Universal Robots PolyScope program: rtde_control_loop.urp

Program rtde_control_loop (installation=default directory=/programs/usbdisk createdIn=3.2.19275 lastSavedIn=0.0.0 robotSerialNumber=20195001564)
Calibrated DH parameters: a=[0.000053, -0.575316, -0.491508, -0.00015, 0.000016, 0]; d=[0.181047, 73.792979, -575.127925, 501.508986, 0.1198, 0.115548]; alpha=[1.570273, 0.002844, 0.000581, 1.569979, -1.569422, 0]; deltaTheta=[-0.000001, 0.349752, 5.398781, 0.534651, 0.000006, 0]
InitVariablesNode
BeforeStart
  setp := Joint_6_name
  SuppressedNode
    Script: rtde_set_watchdog("input_int_register_0", 1, "PAUSE")
Robot Program (runOnlyOnce=false)
  Script: write_output_integer_register(0, 0)
  Wait Sleep waitTime=0.01
  MoveL speed 250 mm/s, acceleration 1200 mm/s^2 (useActiveTCP=true) feature=Base
    Waypoint Variable (Variable): variable=setp
  Script: write_output_integer_register(0, 1)
  Wait Sleep waitTime=0.01
Thread Thread_1 (runOnlyOnce=false)
  setp := Joint_6_name
  Loop Forever
    tmp := p[0,0,0,0,0,0]
    Script: tmp[0] = read_input_float_register(0)
    Script: tmp[1] = read_input_float_register(1)
    Script: tmp[2] = read_input_float_register(2)
    Script: tmp[3] = read_input_float_register(3)
    Script: tmp[4] = read_input_float_register(4)
    Script: tmp[5] = read_input_float_register(5)
    If tmp != p[0,0,0,0,0,0]
      setp := tmp
    Script: sync()
